{attribute addProperty BoxType "EK1100-0000-0018"}
{attribute addProperty Id "Beckhoff_EL66xxEK1122Beckhoff_EL66xxEK1122_25FC55822184273A_0001_EL6601_0000_0000EL6601_194A340D8010A_0002_EL6601_0000_0001EL6601_194A340D8010A_0003_EL6601_0000_0016EL6601_194A340D8010A_0004_EL6601_0000_0017EL6601_194A340D8010A_0005_EL6601_0000_0018EL6601_194A340D8010A_0006_EL6601_0000_0019EL6601_194A340D8010A_0007_EL6601_0000_0021EL6601_194A340D8010A_0008_EL6614_0000_0016EL6614_194A340D8010A_0009_EL6614_0000_0017EL6614_194A340D8010A_0010_EL6614_0000_0018EL6614_194A340D8010A_0011_EL6614_0000_0019EL6614_194A340D8010A_0012_EL6614_0000_0021EL6614_194A340D8010A_0013_EL6631_0000_0016EL6631_8C99EE5012816A_0014_EL6631_0000_0017EL6631_8C99EE5012816A_0015_EL6631_0000_0018EL6631_8C99EE5012816A_0016_EL6631_0010_0016EL6631_8C99EE5012816A_0017_EL6631_0010_0017EL6631_8C99EE5012816A_0018_EL6631_0010_0018EL6631_8C99EE5012816A_0019_EL6652_0000_0017EL6652_8C99EE5012816A_0020_EL6652_0000_0018EL6652_8C99EE5012816A_0021_EL6652_0010_0017EL6652_8C99EE5012816A_0022_EL6652_0010_0018EL6652_8C99EE5012816A_0023_EL6688_0000_0016EL6688_357CAB1619224A_0024_EL6688_0000_0017EL6688_8282893D35244A_0025_EL6688_0000_0018EL6688_8282893D35244A_0026_EL6688_0000_0019EL6688_8282893D35244A_0027_EL6688_0000_0020EL6688_8282893D35244A_0028_EL6688_0000_0022EL6688_7BDEAC9235244A_0029_EL6690_0001_0000EL6690_108834A410413A_0030_EL6690_0001_0016EL6690_108834A410413A_0031_EL6690_0001_0017EL6690_108834A410413A_0037_EL6692_0000_0016EL6692_9D416E6E19224A_0038_EL6692_0000_0017EL6692_9D416E6E19224A_0039_EL6692_0000_0018EL6692_F60FD70919224A_0045_EL6695_0000_0001EL6695_330819D616821A_0047_EL6695_0000_0002EL6695_330819D616821A_0049_EL6695_0000_0003EL6695_330819D616821A_0051_EL6695_0000_0004EL6695_952642F616821A_0053_EL6695_0000_0005EL6695_952642F616821A_0055_EL6695_0000_0006EL6695_952642F616821"}
{attribute addProperty CRC "3184141657"}
{attribute addProperty SizeInBites "8272"}
{attribute addProperty SizeInBytes "1034"}
TYPE Beckhoff_EL66xx_BDCA2559 EXTENDS EK1100_179A0949 :
STRUCT
	{attribute addProperty Name "Beckhoff_EL66xxEK1122"}
	Beckhoff_EL66xxEK1122 : Beckhoff_EL66xxEK1122_25FC5582;
	{attribute addProperty Name "A_0001_EL6601_0000_0000"}
	A_0001_EL6601_0000_0000 : EL6601_194A340D;
	{attribute addProperty Name "A_0002_EL6601_0000_0001"}
	A_0002_EL6601_0000_0001 : EL6601_194A340D;
	{attribute addProperty Name "A_0003_EL6601_0000_0016"}
	A_0003_EL6601_0000_0016 : EL6601_194A340D;
	{attribute addProperty Name "A_0004_EL6601_0000_0017"}
	A_0004_EL6601_0000_0017 : EL6601_194A340D;
	{attribute addProperty Name "A_0005_EL6601_0000_0018"}
	A_0005_EL6601_0000_0018 : EL6601_194A340D;
	{attribute addProperty Name "A_0006_EL6601_0000_0019"}
	A_0006_EL6601_0000_0019 : EL6601_194A340D;
	{attribute addProperty Name "A_0007_EL6601_0000_0021"}
	A_0007_EL6601_0000_0021 : EL6601_194A340D;
	{attribute addProperty Name "A_0008_EL6614_0000_0016"}
	A_0008_EL6614_0000_0016 : EL6614_194A340D;
	{attribute addProperty Name "A_0009_EL6614_0000_0017"}
	A_0009_EL6614_0000_0017 : EL6614_194A340D;
	{attribute addProperty Name "A_0010_EL6614_0000_0018"}
	A_0010_EL6614_0000_0018 : EL6614_194A340D;
	{attribute addProperty Name "A_0011_EL6614_0000_0019"}
	A_0011_EL6614_0000_0019 : EL6614_194A340D;
	{attribute addProperty Name "A_0012_EL6614_0000_0021"}
	A_0012_EL6614_0000_0021 : EL6614_194A340D;
	{attribute addProperty Name "A_0013_EL6631_0000_0016"}
	A_0013_EL6631_0000_0016 : EL6631_8C99EE50;
	{attribute addProperty Name "A_0014_EL6631_0000_0017"}
	A_0014_EL6631_0000_0017 : EL6631_8C99EE50;
	{attribute addProperty Name "A_0015_EL6631_0000_0018"}
	A_0015_EL6631_0000_0018 : EL6631_8C99EE50;
	{attribute addProperty Name "A_0016_EL6631_0010_0016"}
	A_0016_EL6631_0010_0016 : EL6631_8C99EE50;
	{attribute addProperty Name "A_0017_EL6631_0010_0017"}
	A_0017_EL6631_0010_0017 : EL6631_8C99EE50;
	{attribute addProperty Name "A_0018_EL6631_0010_0018"}
	A_0018_EL6631_0010_0018 : EL6631_8C99EE50;
	{attribute addProperty Name "A_0019_EL6652_0000_0017"}
	A_0019_EL6652_0000_0017 : EL6652_8C99EE50;
	{attribute addProperty Name "A_0020_EL6652_0000_0018"}
	A_0020_EL6652_0000_0018 : EL6652_8C99EE50;
	{attribute addProperty Name "A_0021_EL6652_0010_0017"}
	A_0021_EL6652_0010_0017 : EL6652_8C99EE50;
	{attribute addProperty Name "A_0022_EL6652_0010_0018"}
	A_0022_EL6652_0010_0018 : EL6652_8C99EE50;
	{attribute addProperty Name "A_0023_EL6688_0000_0016"}
	A_0023_EL6688_0000_0016 : EL6688_357CAB16;
	{attribute addProperty Name "A_0024_EL6688_0000_0017"}
	A_0024_EL6688_0000_0017 : EL6688_8282893D;
	{attribute addProperty Name "A_0025_EL6688_0000_0018"}
	A_0025_EL6688_0000_0018 : EL6688_8282893D;
	{attribute addProperty Name "A_0026_EL6688_0000_0019"}
	A_0026_EL6688_0000_0019 : EL6688_8282893D;
	{attribute addProperty Name "A_0027_EL6688_0000_0020"}
	A_0027_EL6688_0000_0020 : EL6688_8282893D;
	{attribute addProperty Name "A_0028_EL6688_0000_0022"}
	A_0028_EL6688_0000_0022 : EL6688_7BDEAC92;
	{attribute addProperty Name "A_0029_EL6690_0001_0000"}
	A_0029_EL6690_0001_0000 : EL6690_108834A4;
	{attribute addProperty Name "A_0030_EL6690_0001_0016"}
	A_0030_EL6690_0001_0016 : EL6690_108834A4;
	{attribute addProperty Name "A_0031_EL6690_0001_0017"}
	A_0031_EL6690_0001_0017 : EL6690_108834A4;
	{attribute addProperty Name "A_0037_EL6692_0000_0016"}
	A_0037_EL6692_0000_0016 : EL6692_9D416E6E;
	{attribute addProperty Name "A_0038_EL6692_0000_0017"}
	A_0038_EL6692_0000_0017 : EL6692_9D416E6E;
	{attribute addProperty Name "A_0039_EL6692_0000_0018"}
	A_0039_EL6692_0000_0018 : EL6692_F60FD709;
	{attribute addProperty Name "A_0045_EL6695_0000_0001"}
	A_0045_EL6695_0000_0001 : EL6695_330819D6;
	{attribute addProperty Name "A_0047_EL6695_0000_0002"}
	A_0047_EL6695_0000_0002 : EL6695_330819D6;
	{attribute addProperty Name "A_0049_EL6695_0000_0003"}
	A_0049_EL6695_0000_0003 : EL6695_330819D6;
	{attribute addProperty Name "A_0051_EL6695_0000_0004"}
	A_0051_EL6695_0000_0004 : EL6695_952642F6;
	{attribute addProperty Name "A_0053_EL6695_0000_0005"}
	A_0053_EL6695_0000_0005 : EL6695_952642F6;
	{attribute addProperty Name "A_0055_EL6695_0000_0006"}
	A_0055_EL6695_0000_0006 : EL6695_952642F6;
END_STRUCT
END_TYPE

(* stored: Version 1.2.0.0, ProductVersion 3.1.4024.9
   DUT Beckhoff_EL66xx_BDCA2559: Id {86ae682e-86c4-444f-9481-2ffd24579940} *)
